PROGRAM MAIN
VAR
	spawnRate: REAL := 2;
	boxSpeed: REAL := 3;
	runBelt: BOOL := TRUE;
	autoDirection: BOOL := TRUE;
	direction: DINT := 0; //0 = left , else = right
	cameraConfig: DINT := 1; //there are 6 camera configurations (from 1 to 6). Other numbers will just run config 1
	
	//To use the water tank. If both fill and unfill have the same value the water will stay still;
	fill: BOOL :=  FALSE; //
	unfill: BOOL := FALSE;
END_VAR

END_PROGRAM

(* stored: Version 1.1.0.1, ProductVersion 3.1.4024.9
   POU MAIN: Id {167e6138-b7c2-4d34-bba2-2fec0da3103c}, SpecialFunc None *)
